FUNCTION_BLOCK BoxRemover
VAR_INPUT
END_VAR
VAR_OUTPUT
END_VAR
VAR
	
	CarriageAtPickUp	:=BOOL;
	CarriageAtDrop := BOOL;
	BoxDropped := BOOL;




END_VAR

END_FUNCTION_BLOCK

(* stored: Version 1.1.0.1, ProductVersion 3.1.4024.2
   POU BoxRemover: Id {96321d4f-7b48-4734-a4b8-a1b61b3a0819}, SpecialFunc None *)
